// TIA Portal project "Com_PLC_Camera" (V16)

(* hardware
DEVICE "Station S7-1200_1"  S7-1200 Station
   slot 0: "Châssis_0"  S7-1200 Rack  Rack  V1.0
   slot 1: "EOLT_Standard"  CPU 1214C DC/DC/Rly  6ES7 214-1HG40-0XB0  V4.4
DEVICE "Appareil GSD_1"  GSD.Device.PN
   slot 0: "Châssis"  Rack  V1.0
   slot 0: "InSight"  In-Sight IS2XXX CC-B  IS2XXX  5.9.1
      slot 0: "In-Sight IS2XXX CC-B"  In-Sight IS2XXX CC-B  5.9.1
      slot 1: "Interface"  Interface
         slot 1: "Port 1"  Port 1
   slot 1: "Contrôle des acquisitions_1"  Acquisition Control  5.9.1
      slot 0: "Contrôle des acquisitions"  Acquisition Control  5.9.1
   slot 2: "État des acquisitions_1"  Acquisition Status  5.9.1
      slot 0: "État des acquisitions"  Acquisition Status  5.9.1
   slot 3: "Contrôle de l'inspection_1"  Inspection Control  5.9.1
      slot 0: "Contrôle de l'inspection"  Inspection Control  5.9.1
   slot 4: "Status du contrôle_1"  Inspection Status  5.9.1
      slot 0: "Status du contrôle"  Inspection Status  5.9.1
   slot 5: "Contrôle de la commande_1"  Command Control  5.9.1
      slot 0: "Contrôle de la commande"  Command Control  5.9.1
   slot 6: "Contrôle des événements Soft_1"  SoftEvent Control  5.9.1
      slot 0: "Contrôle des événements Soft"  SoftEvent Control  5.9.1
   slot 7: "Données utilisateur - 64 octets_1"  User Data - 64 bytes  5.9.1
      slot 0: "Données utilisateur - 64 octets"  User Data - 64 bytes  5.9.1
   slot 8: "Résultats - 64 octets_1"  Results - 64 bytes  5.9.1
      slot 0: "Résultats - 64 octets"  Results - 64 bytes  5.9.1
DEVICE "Appareil GSD_3"  GSD.Device.PN
   slot 0: "Châssis"  Rack  V1.0
   slot 0: "IV"  IV2-G30*  IV2-G30*  1.0
      slot 0: "IV2-G30*"  IV2-G30*  1.0
      slot 1: "Interface"  Interface
         slot 1: "Port 1"  Port 1
   slot 1: "Command Control_1"  Command Control
      slot 0: "Command Control"  Command Control
   slot 2: "Command Status Bits_1"  Command Status Bits
      slot 0: "Command Status Bits"  Command Status Bits
   slot 3: "Device Result Bits_1"  Device Result Bits
      slot 0: "Device Result Bits"  Device Result Bits
   slot 4: "Device Status Words_1"  Device Status Words
      slot 0: "Device Status Words"  Device Status Words
   slot 5: "Device Statistics_1"  Device Statistics
      slot 0: "Device Statistics"  Device Statistics
   slot 6: "Position Adjust Result_1"  Position Adjust Result
      slot 0: "Position Adjust Result"  Position Adjust Result
   slot 7: "Tool Result_1"  Tool Result
      slot 0: "Tool Result"  Tool Result
   slot 8: "Tool Result_2"  Tool Result
      slot 0: "Tool Result"  Tool Result
   slot 9: "Tool Result_3"  Tool Result
      slot 0: "Tool Result"  Tool Result
DEVICE "Appareil GSD_2"  GSD.Device.PN
   slot 0: "Châssis"  Rack  V1.0
   slot 0: "DataMan"  DataMan 200  DMR-200#-00
      slot 0: "DataMan 200"  DataMan 200
      slot 1: "Interface"  Interface
         slot 1: "Port_1"  Port
   slot 1: "Contrôle de l'acquisition_1"  Acquisition Control
      slot 0: "Contrôle de l'acquisition"  Acquisition Control
   slot 2: "État de l'acquisition_1"  Acquisition Status
      slot 0: "État de l'acquisition"  Acquisition Status
   slot 3: "Contrôle des résultats_1"  Results Control
      slot 0: "Contrôle des résultats"  Results Control
   slot 4: "État des résultats_1"  Results Status
      slot 0: "État des résultats"  Results Status
   slot 5: "Contrôle des événements apériodiques_1"  Soft Event Control
      slot 0: "Contrôle des événements apériodiques"  Soft Event Control
   slot 6: "Données utilisateur - 64 octets_1"  User Data - 64 bytes
      slot 0: "Données utilisateur - 64 octets"  User Data - 64 bytes
   slot 7: "Données des résult. - 64 octets_1"  Result Data - 64 bytes
      slot 0: "Données des résult. - 64 octets"  Result Data - 64 bytes
*)

// ===== PLC "EOLT_Standard"  CPU 1214C DC/DC/Rly =====

VAR_GLOBAL   // PLC tag table "Table de variables standard"
   "System_Byte" AT %MB1 : Byte;
   "FirstScan" AT %M1.0 : Bool;
   "DiagStatusUpdate" AT %M1.1 : Bool;
   "AlwaysTRUE" AT %M1.2 : Bool;
   "AlwaysFALSE" AT %M1.3 : Bool;
   "Clock_Byte" AT %MB0 : Byte;
   "Clock_10Hz" AT %M0.0 : Bool;
   "Clock_5Hz" AT %M0.1 : Bool;
   "Clock_2.5Hz" AT %M0.2 : Bool;
   "Clock_2Hz" AT %M0.3 : Bool;
   "Clock_1.25Hz" AT %M0.4 : Bool;
   "Clock_1Hz" AT %M0.5 : Bool;
   "Clock_0.625Hz" AT %M0.6 : Bool;
   "Clock_0.5Hz" AT %M0.7 : Bool;
   "Tag_1" AT %M4.0 : Bool;
   "Tag_2" AT %Q0.5 : Bool;
   "Tag_3" AT %QW0 : Int;
END_VAR

VAR_GLOBAL   // PLC tag table "KeyenceIV2_tags"
   "IV2_TriggerResponse" AT %I200.0 : Bool;
   "IV2_Busy" AT %I202.2 : Bool;
   "IV2_Run" AT %I202.4 : Bool;
   "IV2_Ready" AT %I202.5 : Bool;
   "IV2_Overall_JudgementOK" AT %I204.0 : Bool;
   "IV2_Tool1_Result" AT %I206.0 : Bool;
   "IV2_Tool2_Result" AT %I206.1 : Bool;
   "IV2_Tool3_Result" AT %I206.2 : Bool;
   "IV2_TriggerRequest" AT %Q200.0 : Bool;
   "ProgramSwitchingRequest" AT %Q200.2 : Bool;
   "WarningClearRequest" AT %Q200.3 : Bool;
   "IV2_TriggerFailed" AT %I201.0 : Bool;
   "IV2_TriggerReady" AT %I202.6 : Bool;
   "IV2_ResultUpdateComplete" AT %I202.1 : Bool;
   "IV2_ResultAvailable" AT %I202.0 : Bool;
   "IV2_Overall judgement_NG" AT %I204.6 : Bool;
END_VAR

ORGANIZATION_BLOCK "Main"   // OB1, LAD, ProgramCycle
TITLE = "Main Program Sweep (Cycle)"
{ S7_Optimized_Access := 'TRUE' }
VERSION : 0.1
   VAR_INPUT
      Initial_Call : Bool;   // Initial call of this OB
      Remanence : Bool;   // =True, if remanent data are available
   END_VAR
BEGIN
END_ORGANIZATION_BLOCK